// TIA Portal V20 export
DATA_BLOCK "Dancer_DB"   // DB190
// stored: InstanceOfName Unit1.Em3.Dancer, InstanceOfType FB, Namespace Unit1.Em3
"Unit1.Em3.Dancer"
   // VAR
   //    instLConSMC_RFG { S7_SetPoint := 'True'} : "LConSMC_RFG";
   // END_VAR
BEGIN
END_DATA_BLOCK
